(*
SPDX-FileCopyrightText: © 2026 Oleksandr Tiutyk <trofimich@gmail.com>
SPDX-License-Identifier: MIT
License: https://opensource.org/license/mit
*)

(*!
<summary>Changes the bound file's position using a configured offset and origin.</summary>
<description>
The resource owner must keep the file acquired through task stopping. Configure Position, Origin and Timeout
before Start and keep them unchanged until STOPPED. Missing binding and native errors use the base Task
failure and cleanup path. Cancellation waits for submitted I/O and does not restore the previous file
position. Reset from STOPPED clears the binding and native request state, preserving offset, origin and
timeout.
</description>
*)

{attribute 'no_explicit_call' := 'do not call this function block directly'}
FUNCTION_BLOCK SetPositionInFile EXTENDS FileContentTask
VAR_STAT
	//! <summary>Static type metadata available before the base task initializes its default name.</summary>
	{attribute 'hide'}
	_ClassName : STRING := __POUNAME();
END_VAR
VAR
    _SetPosition : Tc2_System.FB_FileSeek;
END_VAR

(*!
<summary>Exposes the native operation target copied from the bound file resource.</summary>
<description>
The resource target overwrites a separately assigned value before native submission. Configure the resource
owner to select a target; do not change this value while the task is running.
</description>
*)
{attribute 'monitoring' := 'call'}
PROPERTY AmsNetId : Tc2_System.T_AmsNetID
GET
AmsNetId := _SetPosition.sNetId;
END_GET
SET
_SetPosition.sNetId := AmsNetId;
END_SET
END_PROPERTY

(*!
<summary>Provides the concrete type name used in diagnostics.</summary>
<description>
Returns borrowed read-only metadata; keep the instance alive and do not modify the referenced string.
Initialized static storage is ready during base Task.FB_init; this getter has no side effects or exceptions.
</description>
*)
{attribute 'monitoring' := 'call'}
PROPERTY ClassName : REFERENCE TO STRING
GET
ClassName REF= _ClassName;
END_GET
END_PROPERTY

(*!
<summary>Reports whether the underlying native file operation is busy.</summary>
<description>
Observes native I/O, including work drained during stopping. FALSE is not a task-success result and does not
independently permit the resource owner to close or destroy the file.
</description>
*)
{attribute 'monitoring' := 'call'}
PROPERTY FileOperationInProgress : BOOL
GET
FileOperationInProgress := _SetPosition.bBusy;
END_GET
END_PROPERTY

(*!
<summary>Provides the library namespace used in diagnostics.</summary>
<description>Returns borrowed read-only namespace storage; do not modify the referenced string.</description>
*)
{attribute 'monitoring' := 'call'}
PROPERTY NamespaceName : REFERENCE TO STRING
GET
NamespaceName REF= CurrentNamespace.Name;
END_GET
END_PROPERTY

(*!
<summary>Clears the borrowed binding and native request state after stopping.</summary>
<description>
Preserves Position, Origin and Timeout. Does not cancel pending I/O; stopping must finish first.
</description>
*)
METHOD PROTECTED OnReset
SUPER^.OnReset();

_SetPosition(bExecute := FALSE);
END_METHOD

(*!
<summary>Changes the position of the bound file using the configured offset and origin.</summary>
<description>
Requires a live bound resource whose owner keeps the handle acquired until stopping completes. Native errors
raise an exception for the base Task failure and cleanup path without dynamic string-builder allocations;
completed I/O effects are not rolled back.
</description>
<param name="processingState">BUSY while pending; DONE after native completion without an error.</param>
<param name="stopReasonMessage">Not changed; native failures use exceptions.</param>
*)
METHOD PROTECTED OnRunning
VAR_OUTPUT
	processingState : TOF_Tasks.TASK_PROCESSING_STATE;
END_VAR
VAR_IN_OUT
	stopReasonMessage : TOF_Core.ERROR_MESSAGE;
END_VAR
VAR
	errorMessage : TOF_Core.ERROR_MESSAGE;
END_VAR
IF NOT _SetPosition.bExecute THEN 
	IF NOT __ISVALIDREF(_FileHandleResource) THEN
		TOF_Core.Exceptions.ThrowDataMemberNotSpecified(
			sourceNamespaceName := NamespaceName,
			sourceClassName := ClassName,
			sourcePOUName := __POUNAME(),
			sourcePosition := __POSITION(),
			dataMemberName := 'FileHandleResource'
		);		
	END_IF
	
	_SetPosition.sNetId := _FileHandleResource.AmsNetId;
	_SetPosition.hFile := _FileHandleResource.FileHandle;
END_IF

_SetPosition(bExecute := TRUE);

IF _SetPosition.bError THEN
	TOF_Core.WideStrings.Append255(
		errorMessage,
		"An error occurred while changing position in file ",
		TO_WSTRING(FilePath),
		"'");

	FileSystemExceptions.ThrowFileSystem(
		sourceNamespaceName := NamespaceName,
		sourceClassName := ClassName,
		sourcePOUName := __POUNAME(),
		sourcePosition := __POSITION(),
		message := errorMessage,
		errorCode := _SetPosition.nErrId
	);
END_IF

IF NOT _SetPosition.bBusy THEN
	processingState := TOF_Tasks.TASK_PROCESSING_STATE.DONE;
END_IF
END_METHOD

(*!
<summary>Wait for an already submitted file operation before allowing handle release.</summary>
<description>
FALSE on bExecute only avoids a new request; it does not abort the pending one. Runs for every stop reason. If
no operation is busy, stopping is ready immediately.
</description>
<param name="readyToRelease">TRUE after pending work has completed and release may begin.</param>
*)

METHOD PROTECTED OnStopping
VAR_OUTPUT
	readyToRelease : BOOL;
END_VAR
IF _SetPosition.bBusy THEN
	_SetPosition(bExecute := FALSE);
END_IF

readyToRelease := NOT _SetPosition.bBusy;
END_METHOD

{attribute 'monitoring' := 'call'}
(*!
<summary>Selects the native reference point for the requested offset.</summary>
<description>
Configure together with Position before Start and keep unchanged until STOPPED. Passed to FB_FileSeek without
additional validation; Reset preserves it.
</description>
*)
PROPERTY Origin : Tc2_System.E_SeekOrigin
GET
Origin := _SetPosition.eOrigin;
END_GET
SET
_SetPosition.eOrigin := Origin;
END_SET
END_PROPERTY

{attribute 'monitoring' := 'call'}
(*!
<summary>Provides the requested native seek offset relative to Origin.</summary>
<description>
This is configuration, not the resulting file position. Set before Start and keep unchanged until STOPPED;
Reset preserves it. Native constraints depend on Origin and the opened file.
</description>
*)
PROPERTY Position : DINT
GET
Position := _SetPosition.nSeekPos;
END_GET
SET
_SetPosition.nSeekPos := Position;
END_SET
END_PROPERTY

(*!
<summary>Reports the size of this concrete instance in bytes.</summary>
*)
{attribute 'monitoring' := 'call'}
PROPERTY SelfSize : ULINT
GET
SelfSize := XSIZEOF(THIS^);
END_GET
END_PROPERTY

(*!
<summary>Configures the timeout passed to native operation requests.</summary>
<description>
Set before Start and keep unchanged until STOPPED. Reset preserves this value. It is not an overall task
deadline or a guarantee of resource release after a timeout.
</description>
*)
{attribute 'monitoring' := 'call'}
PROPERTY Timeout : TIME
GET
Timeout := _SetPosition.tTimeout;
END_GET
SET
_SetPosition.tTimeout := Timeout;
END_SET
END_PROPERTY

END_FUNCTION_BLOCK

(* stored: Version 1.1.0.1
   POU SetPositionInFile: Id {2ffd7f2a-d3d6-47c9-9d3a-1e9a401c5b19}, SpecialFunc None
   Folder Inputs: Id {a5df2b6b-917f-4f8c-b00d-1f6201a63ac9}
   Folder Overriden methods: Id {e0bbb6ab-3610-477a-8601-1e6464605dbf}
   Property AmsNetId: Id {962933ed-c3fb-407a-924b-c22895e6ca9b}
   Get Get: Id {fd9fa5cf-c7af-48b9-ae46-81212e5af96f}
   Set Set: Id {63cff82e-1299-472d-b0f6-34d2d19d5720}
   Property ClassName: Id {cfdb6426-d476-42b9-99d1-4f5358e336a0}
   Get Get: Id {9308678a-bfc7-4c39-9bf3-a53309e5994e}
   Property FileOperationInProgress: Id {d2f9cbc9-0bf1-4bfb-bb02-4e28ad125b5c}
   Get Get: Id {2f0a7120-515d-4b95-a71e-21856b7a972c}
   Property NamespaceName: Id {5d4e917a-caa7-42e6-b306-afda1ea469d1}
   Get Get: Id {14add75a-a1cd-47cc-8e51-098a619ad651}
   Method OnReset: Id {cfc6df6b-d281-4a15-b319-5749c80fbdb9}
   Method OnRunning: Id {5baa2eff-208e-451f-9d4c-98409c9ff39d}
   Method OnStopping: Id {a3832dc5-33f8-4a9b-9737-37bc7f72bd87}
   Property Origin: Id {59a9a4c8-934e-41d3-b102-8ce67e140be5}
   Get Get: Id {aff431bd-6656-46a8-836e-c5952078887b}
   Set Set: Id {e5a42079-3800-4fef-badd-149a0f68983e}
   Property Position: Id {8bf26b09-787c-4098-a51e-a06a2a359eaa}
   Get Get: Id {335fe352-4856-40ef-bb0c-554974e6ff67}
   Set Set: Id {58209566-1197-4dd9-947a-57418722e8fc}
   Property SelfSize: Id {c9813391-742f-48f8-bb85-0f5cf528183c}
   Get Get: Id {d49aef89-2950-4f78-a37e-432539dcc989}
   Property Timeout: Id {860a0249-7acd-4b02-8556-575cc6a54120}
   Get Get: Id {92bb4a91-5a5d-40f1-a1f2-bce74a7e6d05}
   Set Set: Id {f2d5d237-0ebd-4438-b8df-16e6514a2323} *)
